Yaskawa INFORM job: X2_29-32(-90,180).JBI

/JOB
//NAME X2_29-32(-90,180)
//POS
///NPOS 300,300,300,19,0,0
///TOOL 0
///POSTYPE PULSE
///PULSE
C00000=2000,-95440,-72516,0,38121,0
C00001=-80443,-95440,-72516,-46202,38121,50067
C00002=-52411,-63190,-65629,-41206,65263,51508
C00003=-73087,-23788,-54178,-20049,70640,39353
C00004=-137855,-58890,-63164,50426,57117,3007
C00005=-121629,-1819,-23267,32035,72941,16834
C00006=-120935,3126,-16373,32060,71231,16611
C00007=-120668,5150,-13541,32087,70531,16512
C00008=-120826,7275,-11699,32150,70554,16454
C00009=-120668,5150,-13541,32087,70531,16512
C00010=-120649,6560,-12069,32112,70369,16472
C00011=-120645,6560,-10825,32251,69714,16277
C00012=-120649,6560,-12069,32112,70369,16472
C00013=-120913,4529,-14922,32082,71075,16573
C00014=-121602,-429,-21862,32048,72802,16805
C00015=-120074,-1541,-23154,10906,71264,22392
C00016=-120462,3262,-16191,11181,69532,22093
C00017=-120612,5232,-13331,11295,68818,21971
C00018=-120770,7357,-11488,11363,68799,21912
C00019=-120612,5232,-13331,11295,68818,21971
C00020=-120702,6360,-12382,11332,68826,21940
C00021=-120699,6356,-11141,11388,68075,21868
C00022=-120702,6360,-12382,11332,68826,21940
C00023=-120555,4389,-15254,11219,69547,22062
C00024=-120172,-412,-22245,10944,71297,22361
C00025=-119941,-49108,-60020,12756,52739,20459
C00026=-119789,-74783,-79746,11606,60570,21449
C00027=-121427,-115493,-86071,-971,23186,13
C00028=-103613,-33005,-61039,-35202,65094,-22685
C00029=-118652,-1130,-18887,-50959,75871,-22344
C00030=-120065,3095,-12579,-50928,73991,-22034
C00031=-120612,5858,-10323,-50783,73711,-22168
C00032=-120794,7716,-8707,-50742,73586,-22192
C00033=-120612,6719,-9575,-50786,73699,-22162
C00034=-120612,6754,-8612,-50907,73330,-21953
C00035=-120612,6719,-9575,-50786,73699,-22162
C00036=-120164,4326,-11494,-50910,73914,-22043
C00037=-118762,92,-17836,-50934,75798,-22362
C00038=-120082,-2017,-23568,-21020,76850,-12939
C00039=-120471,2786,-16617,-21041,75059,-12760
C00040=-120621,6055,-13261,-21027,74660,-12744
C00041=-120866,7545,-11965,-20950,74569,-12818
C00042=-120698,6523,-12855,-21003,74632,-12768
C00043=-120698,6506,-12245,-21039,74273,-12705
C00044=-120698,6523,-12855,-21003,74632,-12768
C00045=-120547,3972,-15593,-21018,75020,-12781
C00046=-120163,-831,-22574,-20994,76828,-12964
C00047=-120068,-2141,-23641,-4094,79360,4817
C00048=-120458,2664,-16692,-4000,77538,4745
C00049=-120609,5664,-13523,-3960,77123,4708
C00050=-120915,7025,-12341,-3868,77081,4605
C00051=-120609,5664,-13523,-3960,77123,4708
C00052=-120609,5646,-12752,-3962,76640,4725
C00053=-120609,5664,-13523,-3960,77123,4708
C00054=-120559,4206,-15421,-3970,77544,4711
C00055=-120175,-595,-22406,-4061,79389,4780
C00056=-120687,14813,-21149,-8531,87328,5298
C00057=-120686,13947,-18988,-8540,85572,5418
C00058=-121162,15330,-17687,-8405,85435,5272
C00059=-120827,14308,-18485,-8500,85444,5381
C00060=-120926,18777,-11948,-23218,84672,-11491
C00061=-120686,12805,-15419,-25390,80631,-12632
C00062=-120686,13423,-17789,-25296,82244,-12980
C00063=-103613,-33005,-61039,-35202,65094,-22685
C00064=-121427,-115493,-86071,-971,23186,13
C00065=-119789,-74783,-79746,11606,60570,21449
C00066=-119941,-49108,-60020,12756,52739,20459
C00067=-120686,14413,-19191,15888,76861,21657
C00068=-120686,13677,-16924,15998,75153,21431
C00069=-120864,13854,-15557,16118,74464,21280
C00070=-120686,13319,-15964,16052,74414,21331
C00071=-120685,12972,2532,58159,63782,21773
C00072=-120685,12849,1627,57961,64053,21984
C00073=-120685,12557,-1021,57383,64873,22611
C00074=-118042,2496,-28680,21493,77866,23942
C00075=-119941,-49108,-60020,12756,52739,20459
C00076=-119789,-74783,-79746,11606,60570,21449
C00077=-121427,-115493,-86071,-971,23186,13
C00078=-103613,-33005,-61039,-35202,65094,-22685
C00079=-134099,37898,13128,-30528,62935,-29291
C00080=-134100,37844,14655,-30775,62096,-29040
C00081=-131820,39720,18358,-33617,61933,-27865
C00082=-133865,38946,16955,-31235,61462,-28734
C00083=-133724,38989,23896,-55752,81870,-5528
C00084=-134106,38309,22847,-57056,83615,-3951
C00085=-130543,37429,19989,-57378,86491,-3781
C00086=-124532,-28339,-37080,2656,37858,63256
C00087=-80443,-95440,-72516,-46202,38121,50067
C00088=-628,-74499,-67639,-57475,89722,72456
C00089=3643,-76224,-106676,19950,71810,76872
C00090=-57022,-39792,-97587,-14580,73098,62715
C00091=-77894,6609,-39652,-10081,68656,55583
C00092=-79326,8848,-34628,-9340,66588,55287
C00093=-79882,9812,-32559,-9051,65763,55166
C00094=-80655,11957,-30643,-8578,65611,54918
C00095=-79882,9812,-32559,-9051,65763,55166
C00096=-80541,11612,-30977,-8647,65649,54954
C00097=-80539,10894,-29907,-8717,64633,55031
C00098=-80541,11612,-30977,-8647,65649,54954
C00099=-79996,10638,-33064,-8931,66478,55073
C00100=-78593,8374,-38132,-9661,68553,55366
C00101=-77879,6415,-39661,-10096,68566,55596
C00102=-79312,8664,-34633,-9354,66499,55298
C00103=-79868,9631,-32562,-9065,65674,55178
C00104=-80642,11778,-30647,-8592,65523,54929
C00105=-79868,9631,-32562,-9065,65674,55178
C00106=-80486,11377,-31039,-8686,65573,54978
C00107=-80483,10662,-29965,-8757,64557,55056
C00108=-80486,11377,-31039,-8686,65573,54978
C00109=-79940,10400,-33127,-8971,66401,55097
C00110=-78534,8129,-38197,-9702,68474,55392
C00111=-80101,2636,-42462,-8765,68121,54914
C00112=-81514,5018,-37368,-8012,66098,54596
C00113=-82062,6036,-35274,-7718,65291,54467
C00114=-82824,8247,-33345,-7247,65177,54218
C00115=-82062,6036,-35274,-7718,65291,54467
C00116=-82687,7884,-33751,-7328,65251,54260
C00117=-82684,7173,-32662,-7390,64223,54326
C00118=-82687,7884,-33751,-7328,65251,54260
C00119=-82150,6860,-35861,-7618,66062,54387
C00120=-80765,4464,-40992,-8359,68092,54701
C00121=-102565,-17528,-58279,5105,67037,47705
C00122=-103540,-14129,-52689,5779,65410,47308
C00123=-103914,-12731,-50412,6044,64755,47149
C00124=-104433,-9984,-48291,6364,64897,46981
C00125=-103914,-12731,-50412,6044,64755,47149
C00126=-104359,-10402,-48741,6314,64954,47009
C00127=-104354,-11138,-47602,6366,63880,46952
C00128=-104359,-10402,-48741,6314,64954,47009
C00129=-103995,-11787,-51026,6054,65619,47167
C00130=-103047,-15149,-56634,5395,67274,47560
C00131=-80233,11979,-33534,-13378,69985,55632
C00132=-80229,10556,-31784,-13533,68226,55836
C00133=-80227,10062,-31089,-13596,67561,55913
C00134=-85904,3072,-37201,-10254,66968,54061
C00135=-91604,-2565,-41777,-6847,66341,52198
C00136=-101176,-9655,-47350,-1032,65699,49019
C00137=-100886,-9155,-48096,-1203,66417,49108
C00138=-100216,-7271,-49632,-1590,68341,49304
C00139=-80300,11336,-32181,-3939,63811,54132
C00140=-80297,10024,-30348,-4003,62013,54196
C00141=-80296,9579,-29637,-4028,61349,54220
C00142=-80356,9883,-29495,-3999,61418,54197
C00143=-80338,10281,-30338,-3972,62137,54177
C00144=-80341,11605,-32161,-3909,63935,54114
C00145=-57022,-39792,-97587,-14580,73098,62715
C00146=-628,-74499,-67639,-57475,89722,72456
C00147=-628,-74499,-67639,-57475,89722,72456
C00148=-616,-75233,-71189,-57531,90735,71761
C00149=3643,-76224,-106674,19950,71813,76873
C00150=-42730,11015,-70691,-38334,96086,2936
C00151=-63606,9545,-60534,-45336,92087,-16638
C00152=-78956,5069,-41799,-36523,82652,-30708
C00153=-79715,8164,-36018,-36343,80767,-30358
C00154=-80007,9457,-33651,-36288,80012,-30216
C00155=-80417,12097,-31285,-36126,79775,-30292
C00156=-80007,9457,-33651,-36288,80012,-30216
C00157=-80344,11698,-31669,-36153,79828,-30282
C00158=-80337,10939,-30633,-36254,78993,-30001
C00159=-80344,11698,-31669,-36153,79828,-30282
C00160=-80059,10405,-34052,-36203,80590,-30428
C00161=-79319,7312,-39869,-36371,82488,-30786
C00162=-78994,5332,-41692,-36502,82694,-30736
C00163=-79751,8420,-35912,-36322,80808,-30385
C00164=-80043,9710,-33546,-36267,80051,-30242
C00165=-80452,12349,-31177,-36105,79813,-30317
C00166=-80043,9710,-33546,-36267,80051,-30242
C00167=-80378,11838,-31671,-36133,79874,-30310
C00168=-80371,11075,-30637,-36233,79039,-30029
C00169=-80378,11838,-31671,-36133,79874,-30310
C00170=-80093,10547,-34052,-36183,80637,-30456
C00171=-79355,7462,-39866,-36352,82536,-30815
C00172=-79090,5824,-41546,-36452,82791,-30803
C00173=-79842,8894,-35770,-36272,80900,-30451
C00174=-80133,10177,-33405,-36216,80142,-30307
C00175=-80539,12815,-31031,-36055,79902,-30380
C00176=-80133,10177,-33405,-36216,80142,-30307
C00177=-80467,12378,-31515,-36079,79989,-30382
C00178=-80461,11606,-30490,-36178,79153,-30101
C00179=-80467,12378,-31515,-36079,79989,-30382
C00180=-80184,11095,-33894,-36130,80753,-30529
C00181=-79450,8031,-39703,-36300,82657,-30890
C00182=-79130,5997,-41490,-36432,82820,-30827
C00183=-79881,9061,-35715,-36251,80928,-30474
C00184=-80171,10342,-33350,-36196,80169,-30330
C00185=-80577,12980,-30974,-36035,79928,-30403
C00186=-80171,10342,-33350,-36196,80169,-30330
C00187=-80499,12601,-31443,-36059,80034,-30409
C00188=-80493,11826,-30422,-36158,79199,-30129
C00189=-80499,12601,-31443,-36059,80034,-30409
C00190=-80216,11321,-33822,-36110,80799,-30556
C00191=-79484,8265,-39628,-36281,82705,-30918
C00192=-80360,13355,-34008,-31162,79863,-31191
C00193=-80358,11846,-32319,-31320,78301,-30757
C00194=-80129,11573,-31352,-31494,77744,-30518
C00195=-80458,11751,-31298,-31342,77685,-30622
C00196=-80398,12063,-32232,-31297,78337,-30782
C00197=-80400,13577,-33916,-31139,79899,-31215
C00198=-80289,11819,-32883,-40833,82428,-30239
C00199=-80286,10439,-31086,-40975,81039,-29694
C00200=-80284,9940,-30341,-41041,80492,-29477
C00201=-80262,9799,-30343,-41055,80447,-29451
C00202=-80245,10226,-31168,-40996,81011,-29666
C00203=-80248,11601,-32971,-40853,82401,-30212
C00204=-66712,19655,-58640,-43457,90055,-24381
C00205=-33423,17994,-60377,-60627,102988,-19600
C00206=-628,-74499,-67639,-57475,89722,-77289
C00207=-111516,-94989,-87682,-11539,41033,-8318
C00208=-107125,-12532,-46236,-32676,64375,-10703
C00209=-119952,37605,6162,-31233,75137,-17424
C00210=-120511,42562,14108,-31354,72919,-17016
C00211=-120728,44654,17433,-31427,72005,-16841
C00212=-120598,46946,19889,-31526,71766,-16719
C00213=-120728,44654,17433,-31427,72005,-16841
C00214=-120690,45788,18679,-31469,71861,-16784
C00215=-120687,45721,19851,-31594,71213,-16595
C00216=-120690,45788,18679,-31469,71861,-16784
C00217=-120474,43679,15324,-31394,72783,-16962
C00218=-119917,38688,7316,-31265,75018,-17376
C00219=-121235,29127,929,-10497,72605,-22385
C00220=-120892,33963,8709,-10768,70384,-22067
C00221=-120760,35995,11952,-10883,69467,-21936
C00222=-120625,38237,14258,-10956,69222,-21864
C00223=-120760,35995,11952,-10883,69467,-21936
C00224=-120657,37146,13206,-10937,69303,-21884
C00225=-120654,37124,14427,-10991,68554,-21813
C00226=-120657,37146,13206,-10937,69303,-21884
C00227=-120788,35099,9935,-10821,70230,-22016
C00228=-121127,30229,2096,-10548,72470,-22335
C00229=-114017,-48711,-62992,-16459,47417,-13874
C00230=-111516,-94989,-87682,-11539,41033,-8318
C00231=-126605,-77887,-93073,32833,63422,15189
C00232=-122507,12852,-43627,17515,100315,22769
C00233=-122731,-562,-19309,51196,76332,22742
C00234=-121309,3590,-13049,51151,74446,22427
C00235=-120759,5312,-10468,51156,73690,22291
C00236=-120602,7442,-8613,51127,73573,22309
C00237=-120759,5312,-10468,51156,73690,22291
C00238=-120666,6547,-9361,51143,73609,22295
C00239=-120662,6597,-8073,51308,73115,22013
C00240=-120666,6547,-9361,51143,73609,22295
C00241=-121212,4820,-11958,51134,74367,22434
C00242=-122622,659,-18251,51172,76257,22758
C00243=-122507,10859,-42333,17402,98575,22516
C00244=-121302,-1391,-23074,21379,77148,13095
C00245=-120901,3377,-16122,21398,75339,12912
C00246=-120747,5333,-13267,21416,74597,12833
C00247=-120590,7459,-11416,21370,74514,12875
C00248=-120747,5333,-13267,21416,74597,12833
C00249=-120673,6521,-12221,21396,74547,12851
C00250=-120670,6504,-10992,21468,73832,12721
C00251=-120673,6521,-12221,21396,74547,12851
C00252=-120826,4563,-15090,21376,75296,12931
C00253=-121222,-206,-22073,21354,77121,13119
C00254=-121314,-1652,-23262,4485,79740,-4708
C00255=-120913,3117,-16316,4391,77900,-4639
C00256=-120758,5074,-13462,4356,77144,-4613
C00257=-120601,7199,-11615,4311,77090,-4561
C00258=-120758,5074,-13462,4356,77144,-4613
C00259=-120661,6618,-12165,4328,77134,-4580
C00260=-120658,6600,-10936,4339,76370,-4606
C00261=-120661,6618,-12165,4328,77134,-4580
C00262=-120814,4660,-15035,4362,77900,-4605
C00263=-121209,-107,-22019,4454,79763,-4672
C00264=-120687,46979,12625,8958,83453,-5452
C00265=-120687,46939,12852,8960,83294,-5464
C00266=-121610,47377,14332,9229,82719,-5809
C00267=-120687,46779,13614,8967,82756,-5503
C00268=-120687,46744,18453,25999,77793,12121
C00269=-120687,46348,16793,25935,78533,12285
C00270=-120687,46750,14296,25811,80109,12635
C00271=-133650,-5326,-40947,35821,67459,4738
C00272=-126605,-79487,-84548,34660,58331,13454
C00273=-111516,-94989,-87682,-11539,41033,-8318
C00274=-114017,-48711,-62992,-16459,47417,-13874
C00275=-117875,8541,-26754,-15356,68464,-18868
C00276=-120687,46680,12303,-15684,74586,-21239
C00277=-120687,46183,14573,-15804,72993,-21028
C00278=-120687,45847,15503,-15862,72274,-20933
C00279=-120687,45820,15711,-15860,72146,-20914
C00280=-120686,46430,31549,-51889,62431,-21622
C00281=-120686,46225,30262,-51616,62867,-21897
C00282=-120686,45862,27317,-50999,63909,-22538
C00283=-117875,8541,-26754,-15356,68464,-18868
C00284=-114017,-48711,-62992,-16459,47417,-13874
C00285=-111516,-94989,-87682,-11539,41033,-8318
C00286=-126605,-79487,-84548,34660,58331,13454
C00287=-133650,-5326,-40947,35821,67459,4738
C00288=-107292,16964,-8341,30286,65218,30077
C00289=-107291,16711,-5651,30703,63668,29626
C00290=-107319,17056,-4163,30899,63039,29427
C00291=-107325,17150,-4064,30903,63037,29424
C00292=-107531,17120,3962,56911,83437,5110
C00293=-107292,16975,3345,57479,84239,4502
C00294=-107292,16775,1094,57407,84952,4997
C00295=-118083,23631,-28824,25815,115568,5891
C00296=-116334,-45445,-82386,24519,90130,1359
C00297=-114916,-111439,-107393,23774,54945,-5331
C00298=-628,-74499,-67639,-57475,89722,-77289
C00299=2000,17994,-60377,0,102988,0
BC00000=30861,666204,744559
BC00001=125925,693938,117612
BC00002=171995,715848,96803
BC00003=199966,729151,84169
BC00004=289373,771673,43785
BC00005=289373,771673,43785
BC00006=289373,771673,43785
BC00007=289373,771673,43785
BC00008=289373,771673,43785
BC00009=289373,771673,43785
BC00010=289373,771673,43785
BC00011=289373,771673,43785
BC00012=289373,771673,43785
BC00013=289373,771673,43785
BC00014=289373,771673,43785
BC00015=275430,758658,78312
BC00016=275430,758658,78312
BC00017=275430,758658,78312
BC00018=275430,758658,78312
BC00019=275430,758658,78312
BC00020=275430,758658,78312
BC00021=275430,758658,78312
BC00022=275430,758658,78312
BC00023=275430,758658,78312
BC00024=275430,758658,78312
BC00025=275430,725446,78312
BC00026=275430,674753,78312
BC00027=160005,679271,117612
BC00028=134493,734471,53
BC00029=134493,734471,53
BC00030=134493,734471,53
BC00031=134493,734471,53
BC00032=134493,734471,53
BC00033=134493,734471,53
BC00034=134493,734471,53
BC00035=134493,734471,53
BC00036=134493,734471,53
BC00037=134493,734471,53
BC00038=120013,731989,63282
BC00039=120013,731989,63282
BC00040=120013,731989,63282
BC00041=120013,731989,63282
BC00042=120013,731989,63282
BC00043=120013,731989,63282
BC00044=120013,731989,63282
BC00045=120013,731989,63282
BC00046=120013,731989,63282
BC00047=143296,743099,87341
BC00048=143296,743099,87341
BC00049=143296,743099,87341
BC00050=143296,743099,87341
BC00051=143296,743099,87341
BC00052=143296,743099,87341
BC00053=143296,743099,87341
BC00054=143296,743099,87341
BC00055=143296,743099,87341
BC00056=160875,733218,0
BC00057=159215,738452,0
BC00058=159050,738970,0
BC00059=154263,739676,0
BC00060=124438,729775,0
BC00061=121804,726587,0
BC00062=123464,721353,0
BC00063=134493,734471,53
BC00064=160005,679271,117612
BC00065=275430,674753,78312
BC00066=275430,725446,78312
BC00067=261630,745054,0
BC00068=261335,750526,0
BC00069=262635,752963,0
BC00070=310200,761264,0
BC00071=269037,768534,0
BC00072=267560,766459,0
BC00073=263869,761272,0
BC00074=263869,761272,0
BC00075=275430,725446,78312
BC00076=275430,674753,78312
BC00077=160005,679271,117612
BC00078=134493,734471,53
BC00079=177141,688062,0
BC00080=175480,693296,0
BC00081=174817,695179,178
BC00082=160472,692881,15
BC00083=152915,732429,1
BC00084=154775,734615,0
BC00085=161011,731782,0
BC00086=160005,693938,117612
BC00087=125925,693938,117612
BC00088=97174,666880,426359
BC00089=199464,674570,1075173
BC00090=48447,721710,1061717
BC00091=196183,770700,1075175
BC00092=196183,770700,1075175
BC00093=196183,770700,1075175
BC00094=196183,770700,1075175
BC00095=196183,770700,1075175
BC00096=196183,770700,1075175
BC00097=196183,770700,1075175
BC00098=196183,770700,1075175
BC00099=196183,770700,1075175
BC00100=196183,770700,1075175
BC00101=139869,760824,1075175
BC00102=139869,760824,1075175
BC00103=139869,760824,1075175
BC00104=139869,760824,1075175
BC00105=139869,760824,1075175
BC00106=139869,760824,1075175
BC00107=139869,760824,1075175
BC00108=139869,760824,1075175
BC00109=139869,760824,1075175
BC00110=139869,760824,1075175
BC00111=15,735270,1075175
BC00112=15,735270,1075175
BC00113=15,735270,1075175
BC00114=15,735270,1075175
BC00115=15,735270,1075175
BC00116=15,735270,1075175
BC00117=15,735270,1075175
BC00118=15,735270,1075175
BC00119=15,735270,1075175
BC00120=15,735270,1075175
BC00121=15,725270,1075175
BC00122=15,725270,1075175
BC00123=15,725270,1075175
BC00124=15,725270,1075175
BC00125=15,725270,1075175
BC00126=15,725270,1075175
BC00127=15,725270,1075175
BC00128=15,725270,1075175
BC00129=15,725270,1075175
BC00130=15,725270,1075175
BC00131=12536,730414,1075175
BC00132=10876,735648,1075175
BC00133=10211,737741,1075175
BC00134=7204,734292,1075175
BC00135=4400,731075,1075175
BC00136=15,726043,1075175
BC00137=15,723950,1075175
BC00138=15,718716,1075175
BC00139=125627,754347,1075175
BC00140=125333,759820,1075175
BC00141=125215,762009,1075175
BC00142=192338,773707,1075173
BC00143=192456,771518,1075175
BC00144=192751,766045,1075175
BC00145=48447,721710,1061717
BC00146=97174,666880,1005640
BC00147=97174,666880,842388
BC00148=97174,666880,900747
BC00149=199464,674570,1075172
BC00150=79996,736581,994878
BC00151=45352,753605,1043201
BC00152=33984,772629,1075175
BC00153=33984,772629,1075175
BC00154=33984,772629,1075175
BC00155=33984,772629,1075175
BC00156=33984,772629,1075175
BC00157=33984,772629,1075175
BC00158=33984,772629,1075175
BC00159=33984,772629,1075175
BC00160=33984,772629,1075175
BC00161=33984,772629,1075175
BC00162=90316,762849,1075175
BC00163=90316,762849,1075175
BC00164=90316,762849,1075175
BC00165=90316,762849,1075175
BC00166=90316,762849,1075175
BC00167=90316,762849,1075175
BC00168=90316,762849,1075175
BC00169=90316,762849,1075175
BC00170=90316,762849,1075175
BC00171=90316,762849,1075175
BC00172=237131,737545,1075175
BC00173=237131,737545,1075175
BC00174=237131,737545,1075175
BC00175=237131,737545,1075175
BC00176=237131,737545,1075175
BC00177=237131,737545,1075175
BC00178=237131,737545,1075175
BC00179=237131,737545,1075175
BC00180=237131,737545,1075175
BC00181=237131,737545,1075175
BC00182=294635,727643,1075175
BC00183=294635,727643,1075175
BC00184=294635,727643,1075175
BC00185=294635,727643,1075175
BC00186=294635,727643,1075175
BC00187=294635,727643,1075175
BC00188=294635,727643,1075175
BC00189=294635,727643,1075175
BC00190=294635,727643,1075175
BC00191=294635,727643,1075175
BC00192=217651,732700,1075175
BC00193=219347,737901,1075175
BC00194=220025,739981,1075175
BC00195=287170,728397,1075175
BC00196=286492,726316,1075175
BC00197=284797,721115,1075175
BC00198=104549,756414,1075175
BC00199=104877,761851,1075175
BC00200=105009,764026,1075175
BC00201=37863,775610,1075175
BC00202=37732,773435,1075175
BC00203=37403,767998,1075175
BC00204=32590,750193,986570
BC00205=32590,674533,986570
BC00206=97174,666880,426359
BC00207=147937,670008,53
BC00208=147937,711773,53
BC00209=147937,730150,53
BC00210=147937,730150,53
BC00211=147937,730150,53
BC00212=147937,730150,53
BC00213=147937,730150,53
BC00214=147937,730150,53
BC00215=147937,730150,53
BC00216=147937,730150,53
BC00217=147937,730150,53
BC00218=147937,730150,53
BC00219=158165,726651,59010
BC00220=158165,726651,59010
BC00221=158165,726651,59010
BC00222=158165,726651,59010
BC00223=158165,726651,59010
BC00224=158165,726651,59010
BC00225=158165,726651,59010
BC00226=158165,726651,59010
BC00227=158165,726651,59010
BC00228=158165,726651,59010
BC00229=154158,704461,35913
BC00230=147937,670008,53
BC00231=303968,673866,53
BC00232=303968,733345,53
BC00233=303968,733345,53
BC00234=303968,733345,53
BC00235=303968,733345,53
BC00236=303968,733345,53
BC00237=303968,733345,53
BC00238=303968,733345,53
BC00239=303968,733345,53
BC00240=303968,733345,53
BC00241=303968,733345,53
BC00242=303968,733345,53
BC00243=303968,733345,53
BC00244=317859,731237,70095
BC00245=317859,731237,70095
BC00246=317859,731237,70095
BC00247=317859,731237,70095
BC00248=317859,731237,70095
BC00249=317859,731237,70095
BC00250=317859,731237,70095
BC00251=317859,731237,70095
BC00252=317859,731237,70095
BC00253=317859,731237,70095
BC00254=294346,742753,94560
BC00255=294346,742753,94560
BC00256=294346,742753,94560
BC00257=294346,742753,94560
BC00258=294346,742753,94560
BC00259=294346,742753,94560
BC00260=294346,742753,94560
BC00261=294346,742753,94560
BC00262=294346,742753,94560
BC00263=294346,742753,94560
BC00264=276740,698523,17248
BC00265=278435,703724,53
BC00266=279113,705804,53
BC00267=283819,705005,53
BC00268=316764,693534,53
BC00269=316086,691453,53
BC00270=314391,686252,53
BC00271=314391,686252,53
BC00272=303968,673866,53
BC00273=147937,670008,53
BC00274=154158,704461,35913
BC00275=166916,707890,15720
BC00276=176272,710404,912
BC00277=176601,715841,53
BC00278=176732,718016,53
BC00279=127735,726480,51
BC00280=162022,730813,53
BC00281=163238,728692,53
BC00282=166278,723391,53
BC00283=166916,707890,15720
BC00284=154158,704461,35913
BC00285=147937,670008,53
BC00286=303968,673866,53
BC00287=314391,686252,53
BC00288=265210,708896,0
BC00289=266905,714097,0
BC00290=267584,716178,0
BC00291=283264,713482,0
BC00292=289747,755484,0
BC00293=287471,755837,0
BC00294=281210,753020,0
BC00295=281210,753020,0
BC00296=281210,753020,0
BC00297=281210,753020,0
BC00298=97174,666880,426359
BC00299=32590,674533,986570
EC00000=-798156,1112951
EC00001=-798156,1112951
EC00002=-798156,1112951
EC00003=-798156,1112951
EC00004=-798156,1112951
EC00005=-798156,1112951
EC00006=-798156,1112951
EC00007=-798156,1112951
EC00008=-798156,1112951
EC00009=-798156,1112951
EC00010=-798156,1112951
EC00011=-798156,1112951
EC00012=-798156,1112951
EC00013=-798156,1112951
EC00014=-798156,1112951
EC00015=-798156,1112951
EC00016=-798156,1112951
EC00017=-798156,1112951
EC00018=-798156,1112951
EC00019=-798156,1112951
EC00020=-798156,1112951
EC00021=-798156,1112951
EC00022=-798156,1112951
EC00023=-798156,1112951
EC00024=-798156,1112951
EC00025=-798156,1112951
EC00026=-798156,1112951
EC00027=-798156,1112951
EC00028=-798156,1112951
EC00029=-798156,1112951
EC00030=-798156,1112951
EC00031=-798156,1112951
EC00032=-798156,1112951
EC00033=-798156,1112951
EC00034=-798156,1112951
EC00035=-798156,1112951
EC00036=-798156,1112951
EC00037=-798156,1112951
EC00038=-798156,1112951
EC00039=-798156,1112951
EC00040=-798156,1112951
EC00041=-798156,1112951
EC00042=-798156,1112951
EC00043=-798156,1112951
EC00044=-798156,1112951
EC00045=-798156,1112951
EC00046=-798156,1112951
EC00047=-798156,1112951
EC00048=-798156,1112951
EC00049=-798156,1112951
EC00050=-798156,1112951
EC00051=-798156,1112951
EC00052=-798156,1112951
EC00053=-798156,1112951
EC00054=-798156,1112951
EC00055=-798156,1112951
EC00056=-798156,1112951
EC00057=-798156,1112951
EC00058=-798156,1112951
EC00059=-798156,1112951
EC00060=-798156,1112951
EC00061=-798156,1112951
EC00062=-798156,1112951
EC00063=-798156,1112951
EC00064=-798156,1112951
EC00065=-798156,1112951
EC00066=-798156,1112951
EC00067=-798156,1112951
EC00068=-798156,1112951
EC00069=-798156,1112951
EC00070=-798156,1112951
EC00071=-798156,1112951
EC00072=-798156,1112951
EC00073=-798156,1112951
EC00074=-798156,1112951
EC00075=-798156,1112951
EC00076=-798156,1112951
EC00077=-798156,1112951
EC00078=-798156,1112951
EC00079=-798156,1112951
EC00080=-798156,1112951
EC00081=-798155,1112951
EC00082=-798156,1112951
EC00083=-798156,1112951
EC00084=-798156,1112951
EC00085=-798156,1112951
EC00086=-798156,1112951
EC00087=-798156,1112951
EC00088=-798156,1112951
EC00089=-798156,1112951
EC00090=-798156,1112951
EC00091=-798156,1112951
EC00092=-798156,1112951
EC00093=-798156,1112951
EC00094=-798156,1112951
EC00095=-798156,1112951
EC00096=-798156,1112951
EC00097=-798156,1112951
EC00098=-798156,1112951
EC00099=-798156,1112951
EC00100=-798156,1112951
EC00101=-798156,1112951
EC00102=-798156,1112951
EC00103=-798156,1112951
EC00104=-798156,1112951
EC00105=-798156,1112951
EC00106=-798156,1112951
EC00107=-798156,1112951
EC00108=-798156,1112951
EC00109=-798156,1112951
EC00110=-798156,1112951
EC00111=-798156,1112951
EC00112=-798156,1112951
EC00113=-798156,1112951
EC00114=-798156,1112951
EC00115=-798156,1112951
EC00116=-798156,1112951
EC00117=-798156,1112951
EC00118=-798156,1112951
EC00119=-798156,1112951
EC00120=-798156,1112951
EC00121=-798156,1112951
EC00122=-798156,1112951
EC00123=-798156,1112951
EC00124=-798156,1112951
EC00125=-798156,1112951
EC00126=-798156,1112951
EC00127=-798156,1112951
EC00128=-798156,1112951
EC00129=-798156,1112951
EC00130=-798156,1112951
EC00131=-798156,1112951
EC00132=-798156,1112951
EC00133=-798156,1112951
EC00134=-798156,1112951
EC00135=-798156,1112951
EC00136=-798156,1112951
EC00137=-798156,1112951
EC00138=-798156,1112951
EC00139=-798156,1112951
EC00140=-798156,1112951
EC00141=-798156,1112951
EC00142=-798155,1112951
EC00143=-798156,1112951
EC00144=-798156,1112951
EC00145=-798156,1112951
EC00146=-798156,1112951
EC00147=-850885,799301
EC00148=-850885,361850
EC00149=-798154,-3
EC00150=-798156,0
EC00151=-798156,0
EC00152=-798156,0
EC00153=-798156,0
EC00154=-798156,0
EC00155=-798156,0
EC00156=-798156,0
EC00157=-798156,0
EC00158=-798156,0
EC00159=-798156,0
EC00160=-798156,0
EC00161=-798156,0
EC00162=-798156,0
EC00163=-798156,0
EC00164=-798156,0
EC00165=-798156,0
EC00166=-798156,0
EC00167=-798156,0
EC00168=-798156,0
EC00169=-798156,0
EC00170=-798156,0
EC00171=-798156,0
EC00172=-798156,0
EC00173=-798156,0
EC00174=-798156,0
EC00175=-798156,0
EC00176=-798156,0
EC00177=-798156,0
EC00178=-798156,0
EC00179=-798156,0
EC00180=-798156,0
EC00181=-798156,0
EC00182=-798156,0
EC00183=-798156,0
EC00184=-798156,0
EC00185=-798156,0
EC00186=-798156,0
EC00187=-798156,0
EC00188=-798156,0
EC00189=-798156,0
EC00190=-798156,0
EC00191=-798156,0
EC00192=-798156,0
EC00193=-798156,0
EC00194=-798156,0
EC00195=-798156,0
EC00196=-798156,0
EC00197=-798156,0
EC00198=-798156,0
EC00199=-798156,0
EC00200=-798156,0
EC00201=-798156,0
EC00202=-798156,0
EC00203=-798156,0
EC00204=-798156,0
EC00205=-798156,0
EC00206=-798156,0
EC00207=-798156,0
EC00208=-798156,0
EC00209=-798156,0
EC00210=-798156,0
EC00211=-798156,0
EC00212=-798156,0
EC00213=-798156,0
EC00214=-798156,0
EC00215=-798156,0
EC00216=-798156,0
EC00217=-798156,0
EC00218=-798156,0
EC00219=-798156,0
EC00220=-798156,0
EC00221=-798156,0
EC00222=-798156,0
EC00223=-798156,0
EC00224=-798156,0
EC00225=-798156,0
EC00226=-798156,0
EC00227=-798156,0
EC00228=-798156,0
EC00229=-798156,0
EC00230=-798156,0
EC00231=-798156,0
EC00232=-798156,0
EC00233=-798156,0
EC00234=-798156,0
EC00235=-798156,0
EC00236=-798156,0
EC00237=-798156,0
EC00238=-798156,0
EC00239=-798156,0
EC00240=-798156,0
EC00241=-798156,0
EC00242=-798156,0
EC00243=-798156,0
EC00244=-798156,0
EC00245=-798156,0
EC00246=-798156,0
EC00247=-798156,0
EC00248=-798156,0
EC00249=-798156,0
EC00250=-798156,0
EC00251=-798156,0
EC00252=-798156,0
EC00253=-798156,0
EC00254=-798156,0
EC00255=-798156,0
EC00256=-798156,0
EC00257=-798156,0
EC00258=-798156,0
EC00259=-798156,0
EC00260=-798156,0
EC00261=-798156,0
EC00262=-798156,0
EC00263=-798156,0
EC00264=-798156,0
EC00265=-798156,0
EC00266=-798156,0
EC00267=-798156,0
EC00268=-798156,0
EC00269=-798156,0
EC00270=-798156,0
EC00271=-798156,0
EC00272=-798156,0
EC00273=-798156,0
EC00274=-798156,0
EC00275=-798156,0
EC00276=-798156,0
EC00277=-798156,0
EC00278=-798156,0
EC00279=-798155,-1
EC00280=-798156,0
EC00281=-798156,0
EC00282=-798156,0
EC00283=-798156,0
EC00284=-798156,0
EC00285=-798156,0
EC00286=-798156,0
EC00287=-798156,0
EC00288=-798156,0
EC00289=-798156,0
EC00290=-798156,0
EC00291=-798156,0
EC00292=-798156,0
EC00293=-798156,0
EC00294=-798156,0
EC00295=-798156,0
EC00296=-798156,0
EC00297=-798156,0
EC00298=-798156,0
EC00299=-798156,0
///POSTYPE BASE
///RECTAN
///RCONF 0,0,0,0,0,0,0,0,0,0,0,0,0,0,0,0,0,0,0,0,0,0,0,0
P00006=0.222,-3.123,-1.508,0.0000,0.0000,0.0000
P00021=-0.225,-6.128,-0.405,0.0000,0.0000,0.0000
P00022=0.222,-3.123,-1.508,0.0000,0.0000,0.0000
P00023=0.143,-0.036,0.682,0.0000,0.0000,0.0000
P00024=0.145,-0.552,1.326,0.0000,0.0000,0.0000
P00025=-2.003,0.006,0.728,0.0000,0.0000,0.0000
P00026=0.562,-0.002,-0.337,0.0000,0.0000,0.0000
P00027=-0.746,0.015,-9.096,0.0000,0.0000,0.0000
P00028=-2.237,-0.018,-7.702,0.0000,0.0000,0.0000
///RCONF 0,0,0,0,1,0,0,0,0,0,0,0,0,0,0,0,0,0,0,0,0,0,0,0
P00033=-0.123,0.612,-5.012,0.0000,0.0000,0.0000
///RCONF 0,0,0,0,0,0,0,0,0,0,0,0,0,0,0,0,0,0,0,0,0,0,0,0
P00034=-0.304,0.773,-2.693,0.0000,0.0000,0.0000
P00035=2.817,0.591,-1.622,0.0000,0.0000,0.0000
P00036=-1.108,-0.829,1.850,0.0000,0.0000,0.0000
P00041=0.192,3.924,0.305,0.0000,0.0000,0.0000
P00042=-0.217,1.941,0.413,0.0000,0.0000,0.0000
P00043=-0.044,-1.937,1.197,0.0000,0.0000,0.0000
P00044=0.687,-2.322,1.156,0.0000,0.0000,0.0000
P00045=-0.068,-0.810,1.603,0.0000,0.0000,0.0000
P00046=0.799,0.043,1.292,0.0000,0.0000,0.0000
//INST
///DATE 2024/04/08 10:40
///ATTR SC,RW
///GROUP1 RB1,BS1
///GROUP2 ST1
NOP
'X2_29-32(-90,180)
MOVJ C00000 BC00000 VJ=100.00  +MOVJ EC00000 VJ=100.00
MOVJ C00001 BC00001 VJ=100.00  +MOVJ EC00001 VJ=100.00
MOVJ C00002 BC00002 VJ=100.00  +MOVJ EC00002 VJ=100.00
MOVJ C00003 BC00003 VJ=100.00  +MOVJ EC00003 VJ=100.00
MOVJ C00004 BC00004 VJ=100.00  +MOVJ EC00004 VJ=100.00
'Path S4862
SFTOF3D
MOVJ C00005 BC00005 VJ=100.00  +MOVJ EC00005 VJ=100.00
MOVL C00006 BC00006 V=800.0  +MOVJ EC00006 VJ=100.00
SMOVL C00007 BC00007 V=166.7  +MOVJ EC00007
SREFP 3 C00008 BC00008  +REFP EC00008
CALL JOB:SEARCH-R1-S13D
SET P042 P006
SFTON3D P042
SMOVL C00009 BC00009 V=166.7  +MOVJ EC00009
SMOVL C00010 BC00010 V=166.7  +MOVJ EC00010
SREFP 3 C00011 BC00011  +REFP EC00011
CALL JOB:SEARCH-R1-S13D
SET P042 P006
SFTON3D P042
SMOVL C00012 BC00012 V=166.7  +MOVJ EC00012
MOVL C00013 BC00013 V=800.0  +MOVJ EC00013 VJ=100.00
MOVL C00014 BC00014 V=1000.0  +MOVJ EC00014 VJ=100.00
'EndPath S4862
'Path S4863
SFTOF3D
MOVJ C00015 BC00015 VJ=100.00  +MOVJ EC00015 VJ=100.00
MOVL C00016 BC00016 V=800.0  +MOVJ EC00016 VJ=100.00
SMOVL C00017 BC00017 V=166.7  +MOVJ EC00017
SREFP 3 C00018 BC00018  +REFP EC00018
CALL JOB:SEARCH-R1-S13D
SET P041 P006
SFTON3D P041
SMOVL C00019 BC00019 V=166.7  +MOVJ EC00019
SMOVL C00020 BC00020 V=166.7  +MOVJ EC00020
SREFP 3 C00021 BC00021  +REFP EC00021
CALL JOB:SEARCH-R1-S13D
SET P041 P006
SFTON3D P041
SMOVL C00022 BC00022 V=166.7  +MOVJ EC00022
MOVL C00023 BC00023 V=800.0  +MOVJ EC00023 VJ=100.00
MOVL C00024 BC00024 V=1000.0  +MOVJ EC00024 VJ=100.00
'EndPath S4863
MOVJ C00025 BC00025 VJ=100.00  +MOVJ EC00025 VJ=100.00
MOVJ C00026 BC00026 VJ=100.00  +MOVJ EC00026 VJ=100.00
MOVJ C00027 BC00027 VJ=100.00  +MOVJ EC00027 VJ=100.00
MOVJ C00028 BC00028 VJ=100.00  +MOVJ EC00028 VJ=100.00
'Path S4864
SFTOF3D
MOVJ C00029 BC00029 VJ=100.00  +MOVJ EC00029 VJ=100.00
MOVL C00030 BC00030 V=800.0  +MOVJ EC00030 VJ=100.00
SMOVL C00031 BC00031 V=166.7  +MOVJ EC00031
SREFP 3 C00032 BC00032  +REFP EC00032
CALL JOB:SEARCH-R1-S13D
SET P045 P006
SFTON3D P045
SMOVL C00033 BC00033 V=166.7  +MOVJ EC00033
SREFP 3 C00034 BC00034  +REFP EC00034
CALL JOB:SEARCH-R1-S13D
SET P045 P006
SFTON3D P045
SMOVL C00035 BC00035 V=166.7  +MOVJ EC00035
MOVL C00036 BC00036 V=800.0  +MOVJ EC00036 VJ=100.00
MOVL C00037 BC00037 V=1000.0  +MOVJ EC00037 VJ=100.00
'EndPath S4864
'Path S4231
SFTOF3D
MOVJ C00038 BC00038 VJ=100.00  +MOVJ EC00038 VJ=100.00
MOVL C00039 BC00039 V=800.0  +MOVJ EC00039 VJ=100.00
SMOVL C00040 BC00040 V=166.7  +MOVJ EC00040
SREFP 3 C00041 BC00041  +REFP EC00041
CALL JOB:SEARCH-R1-S13D
SET P022 P006
SFTON3D P022
SMOVL C00042 BC00042 V=166.7  +MOVJ EC00042
SREFP 3 C00043 BC00043  +REFP EC00043
CALL JOB:SEARCH-R1-S13D
SET P022 P006
SFTON3D P022
SMOVL C00044 BC00044 V=166.7  +MOVJ EC00044
MOVL C00045 BC00045 V=800.0  +MOVJ EC00045 VJ=100.00
MOVL C00046 BC00046 V=1000.0  +MOVJ EC00046 VJ=100.00
'EndPath S4231
'Path S4232
SFTOF3D
MOVJ C00047 BC00047 VJ=100.00  +MOVJ EC00047 VJ=100.00
MOVL C00048 BC00048 V=800.0  +MOVJ EC00048 VJ=100.00
SMOVL C00049 BC00049 V=166.7  +MOVJ EC00049
SREFP 3 C00050 BC00050  +REFP EC00050
CALL JOB:SEARCH-R1-S13D
SET P021 P006
SFTON3D P021
SMOVL C00051 BC00051 V=166.7  +MOVJ EC00051
SREFP 3 C00052 BC00052  +REFP EC00052
CALL JOB:SEARCH-R1-S13D
SET P021 P006
SFTON3D P021
SMOVL C00053 BC00053 V=166.7  +MOVJ EC00053
MOVL C00054 BC00054 V=800.0  +MOVJ EC00054 VJ=100.00
MOVL C00055 BC00055 V=1000.0  +MOVJ EC00055 VJ=100.00
'EndPath S4232
'Path W4886
SFTOF3D
SFTON3D P021
MOVJ C00056 BC00056 VJ=100.00  +MOVJ EC00056 VJ=100.00
SMOVL C00057 BC00057 V=800.0  +MOVJ EC00057
SMOVL C00058 BC00058 V=150.0 PL=0  +MOVJ EC00058
MACRO1 MJ#(0) ARGF6
ARCON
SMOVL C00059 BC00059 V=8.3  +MOVJ EC00059
SFTON3D P022
SMOVL C00060 BC00060 V=8.3  +MOVJ EC00060
ARCOF
SMOVL C00061 BC00061 V=800.0  +MOVJ EC00061
SMOVL C00062 BC00062 V=1000.0  +MOVJ EC00062
SFTOF3D
'EndPath W4886
MOVJ C00063 BC00063 VJ=100.00  +MOVJ EC00063 VJ=100.00
MOVJ C00064 BC00064 VJ=100.00  +MOVJ EC00064 VJ=100.00
MOVJ C00065 BC00065 VJ=100.00  +MOVJ EC00065 VJ=100.00
MOVJ C00066 BC00066 VJ=100.00  +MOVJ EC00066 VJ=100.00
'Path W4887
SFTOF3D
SFTON3D P041
MOVJ C00067 BC00067 VJ=100.00  +MOVJ EC00067 VJ=100.00
SMOVL C00068 BC00068 V=800.0  +MOVJ EC00068
SMOVL C00069 BC00069 V=150.0 PL=0  +MOVJ EC00069
ARCON
SMOVL C00070 BC00070 V=8.3  +MOVJ EC00070
SFTON3D P042
SMOVL C00071 BC00071 V=8.3  +MOVJ EC00071
ARCOF
SMOVL C00072 BC00072 V=800.0  +MOVJ EC00072
SMOVL C00073 BC00073 V=1000.0  +MOVJ EC00073
SFTOF3D
'EndPath W4887
MOVJ C00074 BC00074 VJ=100.00  +MOVJ EC00074 VJ=100.00
MOVJ C00075 BC00075 VJ=100.00  +MOVJ EC00075 VJ=100.00
MOVJ C00076 BC00076 VJ=100.00  +MOVJ EC00076 VJ=100.00
MOVJ C00077 BC00077 VJ=100.00  +MOVJ EC00077 VJ=100.00
MOVJ C00078 BC00078 VJ=100.00  +MOVJ EC00078 VJ=100.00
'Path W4887
SFTOF3D
SFTON3D P045
MOVJ C00079 BC00079 VJ=100.00  +MOVJ EC00079 VJ=100.00
SMOVL C00080 BC00080 V=800.0  +MOVJ EC00080
SMOVL C00081 BC00081 V=150.0 PL=0  +MOVJ EC00081
ARCON
SMOVL C00082 BC00082 V=8.3  +MOVJ EC00082
SMOVL C00083 BC00083 V=8.3  +MOVJ EC00083
ARCOF
SMOVL C00084 BC00084 V=800.0  +MOVJ EC00084
SMOVL C00085 BC00085 V=1000.0  +MOVJ EC00085
SFTOF3D
'EndPath W4887
MOVJ C00086 BC00086 VJ=100.00  +MOVJ EC00086 VJ=100.00
MOVJ C00087 BC00087 VJ=100.00  +MOVJ EC00087 VJ=100.00
MOVJ C00088 BC00088 VJ=100.00  +MOVJ EC00088 VJ=100.00
'R-L Trip
MOVJ C00089 BC00089 VJ=100.00  +MOVJ EC00089 VJ=100.00
CALL JOB:CLEAN-R1_KM_NEW
'WireCut
MOVJ C00090 BC00090 VJ=100.00  +MOVJ EC00090 VJ=100.00
'Path S4234
SFTOF3D
MOVJ C00091 BC00091 VJ=100.00  +MOVJ EC00091 VJ=100.00
MOVL C00092 BC00092 V=800.0  +MOVJ EC00092 VJ=100.00
SMOVL C00093 BC00093 V=166.7  +MOVJ EC00093
SREFP 3 C00094 BC00094  +REFP EC00094
CALL JOB:SEARCH-R1-S13D
SET P034 P006
SFTON3D P034
SMOVL C00095 BC00095 V=166.7  +MOVJ EC00095
SMOVL C00096 BC00096 V=166.7  +MOVJ EC00096
SREFP 3 C00097 BC00097  +REFP EC00097
CALL JOB:SEARCH-R1-S13D
SET P034 P006
SFTON3D P034
SMOVL C00098 BC00098 V=166.7  +MOVJ EC00098
MOVL C00099 BC00099 V=800.0  +MOVJ EC00099 VJ=100.00
MOVL C00100 BC00100 V=1000.0  +MOVJ EC00100 VJ=100.00
'EndPath S4234
'Path S4235
SFTOF3D
MOVJ C00101 BC00101 VJ=100.00  +MOVJ EC00101 VJ=100.00
MOVL C00102 BC00102 V=800.0  +MOVJ EC00102 VJ=100.00
SMOVL C00103 BC00103 V=166.7  +MOVJ EC00103
SREFP 3 C00104 BC00104  +REFP EC00104
CALL JOB:SEARCH-R1-S13D
SET P033 P006
SFTON3D P033
SMOVL C00105 BC00105 V=166.7  +MOVJ EC00105
SMOVL C00106 BC00106 V=166.7  +MOVJ EC00106
SREFP 3 C00107 BC00107  +REFP EC00107
CALL JOB:SEARCH-R1-S13D
SET P033 P006
SFTON3D P033
SMOVL C00108 BC00108 V=166.7  +MOVJ EC00108
MOVL C00109 BC00109 V=800.0  +MOVJ EC00109 VJ=100.00
MOVL C00110 BC00110 V=1000.0  +MOVJ EC00110 VJ=100.00
'EndPath S4235
'Path S4236
SFTOF3D
MOVJ C00111 BC00111 VJ=100.00  +MOVJ EC00111 VJ=100.00
MOVL C00112 BC00112 V=800.0  +MOVJ EC00112 VJ=100.00
SMOVL C00113 BC00113 V=166.7  +MOVJ EC00113
SREFP 3 C00114 BC00114  +REFP EC00114
CALL JOB:SEARCH-R1-S13D
SET P024 P006
SFTON3D P024
SMOVL C00115 BC00115 V=166.7  +MOVJ EC00115
SMOVL C00116 BC00116 V=166.7  +MOVJ EC00116
SREFP 3 C00117 BC00117  +REFP EC00117
CALL JOB:SEARCH-R1-S13D
SET P024 P006
SFTON3D P024
SMOVL C00118 BC00118 V=166.7  +MOVJ EC00118
MOVL C00119 BC00119 V=800.0  +MOVJ EC00119 VJ=100.00
MOVL C00120 BC00120 V=1000.0  +MOVJ EC00120 VJ=100.00
'EndPath S4236
'Path S4237
SFTOF3D
MOVJ C00121 BC00121 VJ=100.00  +MOVJ EC00121 VJ=100.00
MOVL C00122 BC00122 V=800.0  +MOVJ EC00122 VJ=100.00
SMOVL C00123 BC00123 V=166.7  +MOVJ EC00123
SREFP 3 C00124 BC00124  +REFP EC00124
CALL JOB:SEARCH-R1-S13D
SET P023 P006
SFTON3D P023
SMOVL C00125 BC00125 V=166.7  +MOVJ EC00125
SMOVL C00126 BC00126 V=166.7  +MOVJ EC00126
SREFP 3 C00127 BC00127  +REFP EC00127
CALL JOB:SEARCH-R1-S13D
SET P023 P006
SFTON3D P023
SMOVL C00128 BC00128 V=166.7  +MOVJ EC00128
MOVL C00129 BC00129 V=800.0  +MOVJ EC00129 VJ=100.00
MOVL C00130 BC00130 V=1000.0  +MOVJ EC00130 VJ=100.00
'EndPath S4237
'nowe
'Path W4903
SFTOF3D
SFTON3D P024
MOVJ C00131 BC00131 VJ=100.00  +MOVJ EC00131 VJ=100.00
SMOVL C00132 BC00132 V=800.0  +MOVJ EC00132
SMOVL C00133 BC00133 V=150.0 PL=0  +MOVJ EC00133
MACRO1 MJ#(0) ARGF14
ARCON
SMOVL C00134 BC00134 V=9.2  +MOVJ EC00134
SFTON3D P023
SMOVL C00135 BC00135 V=9.2  +MOVJ EC00135
SMOVL C00136 BC00136 V=9.2  +MOVJ EC00136
ARCOF
SMOVL C00137 BC00137 V=800.0  +MOVJ EC00137
SMOVL C00138 BC00138 V=1000.0  +MOVJ EC00138
SFTOF3D
'EndPath W4903
'Path W4906
SFTOF3D
SFTON3D P033
MOVJ C00139 BC00139 VJ=100.00  +MOVJ EC00139 VJ=100.00
SMOVL C00140 BC00140 V=800.0  +MOVJ EC00140
SMOVL C00141 BC00141 V=150.0 PL=0  +MOVJ EC00141
ARCON
SFTON3D P034
SMOVL C00142 BC00142 V=10.7  +MOVJ EC00142
ARCOF
SMOVL C00143 BC00143 V=800.0  +MOVJ EC00143
SMOVL C00144 BC00144 V=1000.0  +MOVJ EC00144
SFTOF3D
'EndPath W4906
MOVJ C00145 BC00145 VJ=100.00  +MOVJ EC00145 VJ=100.00
'WireCut
MOVJ C00146 BC00146 VJ=100.00  +MOVJ EC00146 VJ=100.00
MOVJ C00147 BC00147 VJ=100.00  +MOVJ EC00147 VJ=100.00
MOVJ C00148 BC00148 VJ=100.00  +MOVJ EC00148 VJ=100.00
MOVJ C00149 BC00149 VJ=100.00  +MOVJ EC00149 VJ=100.00
CALL JOB:CLEAN-R1_KM_NEW
MOVJ C00150 BC00150 VJ=100.00  +MOVJ EC00150 VJ=100.00
MOVJ C00151 BC00151 VJ=100.00  +MOVJ EC00151 VJ=100.00
'L-R Trip
'Path S4249
SFTOF3D
MOVJ C00152 BC00152 VJ=100.00  +MOVJ EC00152 VJ=100.00
MOVL C00153 BC00153 V=800.0  +MOVJ EC00153 VJ=100.00
SMOVL C00154 BC00154 V=166.7  +MOVJ EC00154
SREFP 3 C00155 BC00155  +REFP EC00155
CALL JOB:SEARCH-R1-S13D
SET P036 P006
SFTON3D P036
SMOVL C00156 BC00156 V=166.7  +MOVJ EC00156
SMOVL C00157 BC00157 V=166.7  +MOVJ EC00157
SREFP 3 C00158 BC00158  +REFP EC00158
CALL JOB:SEARCH-R1-S13D
SET P036 P006
SFTON3D P036
SMOVL C00159 BC00159 V=166.7  +MOVJ EC00159
MOVL C00160 BC00160 V=800.0  +MOVJ EC00160 VJ=100.00
MOVL C00161 BC00161 V=1000.0  +MOVJ EC00161 VJ=100.00
'EndPath S4249
'Path S4250
SFTOF3D
MOVJ C00162 BC00162 VJ=100.00  +MOVJ EC00162 VJ=100.00
MOVL C00163 BC00163 V=800.0  +MOVJ EC00163 VJ=100.00
SMOVL C00164 BC00164 V=166.7  +MOVJ EC00164
SREFP 3 C00165 BC00165  +REFP EC00165
CALL JOB:SEARCH-R1-S13D
SET P035 P006
SFTON3D P035
SMOVL C00166 BC00166 V=166.7  +MOVJ EC00166
SMOVL C00167 BC00167 V=166.7  +MOVJ EC00167
SREFP 3 C00168 BC00168  +REFP EC00168
CALL JOB:SEARCH-R1-S13D
SET P035 P006
SFTON3D P035
SMOVL C00169 BC00169 V=166.7  +MOVJ EC00169
MOVL C00170 BC00170 V=800.0  +MOVJ EC00170 VJ=100.00
MOVL C00171 BC00171 V=1000.0  +MOVJ EC00171 VJ=100.00
'EndPath S4250
'Path S4251
SFTOF3D
MOVJ C00172 BC00172 VJ=100.00  +MOVJ EC00172 VJ=100.00
MOVL C00173 BC00173 V=800.0  +MOVJ EC00173 VJ=100.00
SMOVL C00174 BC00174 V=166.7  +MOVJ EC00174
SREFP 3 C00175 BC00175  +REFP EC00175
CALL JOB:SEARCH-R1-S13D
SET P026 P006
SFTON3D P026
SMOVL C00176 BC00176 V=166.7  +MOVJ EC00176
SMOVL C00177 BC00177 V=166.7  +MOVJ EC00177
SREFP 3 C00178 BC00178  +REFP EC00178
CALL JOB:SEARCH-R1-S13D
SET P026 P006
SFTON3D P026
SMOVL C00179 BC00179 V=166.7  +MOVJ EC00179
MOVL C00180 BC00180 V=800.0  +MOVJ EC00180 VJ=100.00
MOVL C00181 BC00181 V=1000.0  +MOVJ EC00181 VJ=100.00
'EndPath S4251
'Path S4252
SFTOF3D
MOVJ C00182 BC00182 VJ=100.00  +MOVJ EC00182 VJ=100.00
MOVL C00183 BC00183 V=800.0  +MOVJ EC00183 VJ=100.00
SMOVL C00184 BC00184 V=166.7  +MOVJ EC00184
SREFP 3 C00185 BC00185  +REFP EC00185
CALL JOB:SEARCH-R1-S13D
SET P025 P006
SFTON3D P025
SMOVL C00186 BC00186 V=166.7  +MOVJ EC00186
SMOVL C00187 BC00187 V=166.7  +MOVJ EC00187
SREFP 3 C00188 BC00188  +REFP EC00188
CALL JOB:SEARCH-R1-S13D
SET P025 P006
SFTON3D P025
SMOVL C00189 BC00189 V=166.7  +MOVJ EC00189
MOVL C00190 BC00190 V=800.0  +MOVJ EC00190 VJ=100.00
MOVL C00191 BC00191 V=1000.0  +MOVJ EC00191 VJ=100.00
'EndPath S4252
'Path W4907
SFTOF3D
SFTON3D P026
MOVJ C00192 BC00192 VJ=100.00  +MOVJ EC00192 VJ=100.00
SMOVL C00193 BC00193 V=800.0  +MOVJ EC00193
SMOVL C00194 BC00194 V=150.0 PL=0  +MOVJ EC00194
ARCON
SFTON3D P025
SMOVL C00195 BC00195 V=11.7  +MOVJ EC00195
ARCOF
SMOVL C00196 BC00196 V=800.0  +MOVJ EC00196
SMOVL C00197 BC00197 V=1000.0  +MOVJ EC00197
SFTOF3D
'EndPath W4907
'Path W4908
SFTOF3D
SFTON3D P035
MOVJ C00198 BC00198 VJ=100.00  +MOVJ EC00198 VJ=100.00
SMOVL C00199 BC00199 V=800.0  +MOVJ EC00199
SMOVL C00200 BC00200 V=150.0 PL=0  +MOVJ EC00200
ARCON
SFTON3D P036
SMOVL C00201 BC00201 V=11.7  +MOVJ EC00201
ARCOF
SMOVL C00202 BC00202 V=800.0  +MOVJ EC00202
SMOVL C00203 BC00203 V=1000.0  +MOVJ EC00203
SFTOF3D
'EndPath W4908
MOVJ C00204 BC00204 VJ=100.00  +MOVJ EC00204 VJ=100.00
MOVJ C00205 BC00205 VJ=100.00  +MOVJ EC00205 VJ=100.00
CALL JOB:CLEAN-R1_KM_NEW
MOVJ C00206 BC00206 VJ=100.00  +MOVJ EC00206 VJ=100.00
MOVJ C00207 BC00207 VJ=100.00  +MOVJ EC00207 VJ=100.00
MOVJ C00208 BC00208 VJ=100.00  +MOVJ EC00208 VJ=100.00
'Path S4888
SFTOF3D
MOVJ C00209 BC00209 VJ=100.00  +MOVJ EC00209 VJ=100.00
MOVL C00210 BC00210 V=800.0  +MOVJ EC00210 VJ=100.00
SMOVL C00211 BC00211 V=166.7  +MOVJ EC00211
SREFP 3 C00212 BC00212  +REFP EC00212
CALL JOB:SEARCH-R1-S13D
SET P044 P006
SFTON3D P044
SMOVL C00213 BC00213 V=166.7  +MOVJ EC00213
SMOVL C00214 BC00214 V=166.7  +MOVJ EC00214
SREFP 3 C00215 BC00215  +REFP EC00215
CALL JOB:SEARCH-R1-S13D
SET P044 P006
SFTON3D P044
SMOVL C00216 BC00216 V=166.7  +MOVJ EC00216
MOVL C00217 BC00217 V=800.0  +MOVJ EC00217 VJ=100.00
MOVL C00218 BC00218 V=1000.0  +MOVJ EC00218 VJ=100.00
'EndPath S4888
'Path S4889
SFTOF3D
MOVJ C00219 BC00219 VJ=100.00  +MOVJ EC00219 VJ=100.00
MOVL C00220 BC00220 V=800.0  +MOVJ EC00220 VJ=100.00
SMOVL C00221 BC00221 V=166.7  +MOVJ EC00221
SREFP 3 C00222 BC00222  +REFP EC00222
CALL JOB:SEARCH-R1-S13D
SET P043 P006
SFTON3D P043
SMOVL C00223 BC00223 V=166.7  +MOVJ EC00223
SMOVL C00224 BC00224 V=166.7  +MOVJ EC00224
SREFP 3 C00225 BC00225  +REFP EC00225
CALL JOB:SEARCH-R1-S13D
SET P043 P006
SFTON3D P043
SMOVL C00226 BC00226 V=166.7  +MOVJ EC00226
MOVL C00227 BC00227 V=800.0  +MOVJ EC00227 VJ=100.00
MOVL C00228 BC00228 V=1000.0  +MOVJ EC00228 VJ=100.00
'EndPath S4889
MOVJ C00229 BC00229 VJ=100.00  +MOVJ EC00229 VJ=100.00
MOVJ C00230 BC00230 VJ=100.00  +MOVJ EC00230 VJ=100.00
MOVJ C00231 BC00231 VJ=100.00  +MOVJ EC00231 VJ=100.00
MOVJ C00232 BC00232 VJ=100.00  +MOVJ EC00232 VJ=100.00
'Path S4899
SFTOF3D
MOVJ C00233 BC00233 VJ=100.00  +MOVJ EC00233 VJ=100.00
MOVL C00234 BC00234 V=800.0  +MOVJ EC00234 VJ=100.00
SMOVL C00235 BC00235 V=166.7  +MOVJ EC00235
SREFP 3 C00236 BC00236  +REFP EC00236
CALL JOB:SEARCH-R1-S13D
SET P046 P006
SFTON3D P046
SMOVL C00237 BC00237 V=166.7  +MOVJ EC00237
SMOVL C00238 BC00238 V=166.7  +MOVJ EC00238
SREFP 3 C00239 BC00239  +REFP EC00239
CALL JOB:SEARCH-R1-S13D
SET P046 P006
SFTON3D P046
SMOVL C00240 BC00240 V=166.7  +MOVJ EC00240
MOVL C00241 BC00241 V=800.0  +MOVJ EC00241 VJ=100.00
MOVL C00242 BC00242 V=1000.0  +MOVJ EC00242 VJ=100.00
'EndPath S4899
MOVJ C00243 BC00243 VJ=100.00  +MOVJ EC00243 VJ=100.00
'Path S4888
SFTOF3D
MOVJ C00244 BC00244 VJ=100.00  +MOVJ EC00244 VJ=100.00
MOVL C00245 BC00245 V=800.0  +MOVJ EC00245 VJ=100.00
SMOVL C00246 BC00246 V=166.7  +MOVJ EC00246
SREFP 3 C00247 BC00247  +REFP EC00247
CALL JOB:SEARCH-R1-S13D
SET P028 P006
SFTON3D P028
SMOVL C00248 BC00248 V=166.7  +MOVJ EC00248
SMOVL C00249 BC00249 V=166.7  +MOVJ EC00249
SREFP 3 C00250 BC00250  +REFP EC00250
CALL JOB:SEARCH-R1-S13D
SET P028 P006
SFTON3D P028
SMOVL C00251 BC00251 V=166.7  +MOVJ EC00251
MOVL C00252 BC00252 V=800.0  +MOVJ EC00252 VJ=100.00
MOVL C00253 BC00253 V=1000.0  +MOVJ EC00253 VJ=100.00
'EndPath S4888
'Path S4889
SFTOF3D
MOVJ C00254 BC00254 VJ=100.00  +MOVJ EC00254 VJ=100.00
MOVL C00255 BC00255 V=800.0  +MOVJ EC00255 VJ=100.00
SMOVL C00256 BC00256 V=166.7  +MOVJ EC00256
SREFP 3 C00257 BC00257  +REFP EC00257
CALL JOB:SEARCH-R1-S13D
SET P027 P006
SFTON3D P027
SMOVL C00258 BC00258 V=166.7  +MOVJ EC00258
SMOVL C00259 BC00259 V=166.7  +MOVJ EC00259
SREFP 3 C00260 BC00260  +REFP EC00260
CALL JOB:SEARCH-R1-S13D
SET P027 P006
SFTON3D P027
SMOVL C00261 BC00261 V=166.7  +MOVJ EC00261
MOVL C00262 BC00262 V=800.0  +MOVJ EC00262 VJ=100.00
MOVL C00263 BC00263 V=1000.0  +MOVJ EC00263 VJ=100.00
'EndPath S4889
'Path W4890
SFTOF3D
SFTON3D P027
MOVJ C00264 BC00264 VJ=100.00  +MOVJ EC00264 VJ=100.00
SMOVL C00265 BC00265 V=800.0  +MOVJ EC00265
SMOVL C00266 BC00266 V=150.0 PL=0  +MOVJ EC00266
MACRO1 MJ#(0) ARGF6
ARCON
SMOVL C00267 BC00267 V=6.7  +MOVJ EC00267
SFTON3D P028
SMOVL C00268 BC00268 V=10.0  +MOVJ EC00268
ARCOF
SMOVL C00269 BC00269 V=800.0  +MOVJ EC00269
SMOVL C00270 BC00270 V=1000.0  +MOVJ EC00270
SFTOF3D
'EndPath W4890
MOVJ C00271 BC00271 VJ=100.00  +MOVJ EC00271 VJ=100.00
MOVJ C00272 BC00272 VJ=100.00  +MOVJ EC00272 VJ=100.00
MOVJ C00273 BC00273 VJ=100.00  +MOVJ EC00273 VJ=100.00
MOVJ C00274 BC00274 VJ=100.00  +MOVJ EC00274 VJ=100.00
MOVJ C00275 BC00275 VJ=100.00  +MOVJ EC00275 VJ=100.00
'Path W4900
SFTOF3D
SFTON3D P043
MOVJ C00276 BC00276 VJ=100.00  +MOVJ EC00276 VJ=100.00
SMOVL C00277 BC00277 V=800.0  +MOVJ EC00277
SMOVL C00278 BC00278 V=150.0 PL=0  +MOVJ EC00278
MACRO1 MJ#(0) ARGF14
ARCON
SFTON3D P044
SMOVL C00279 BC00279 V=10.0  +MOVJ EC00279
SMOVL C00280 BC00280 V=10.0  +MOVJ EC00280
ARCOF
SMOVL C00281 BC00281 V=800.0  +MOVJ EC00281
SMOVL C00282 BC00282 V=1000.0  +MOVJ EC00282
SFTOF3D
'EndPath W4900
MOVJ C00283 BC00283 VJ=100.00  +MOVJ EC00283 VJ=100.00
MOVJ C00284 BC00284 VJ=100.00  +MOVJ EC00284 VJ=100.00
MOVJ C00285 BC00285 VJ=100.00  +MOVJ EC00285 VJ=100.00
MOVJ C00286 BC00286 VJ=100.00  +MOVJ EC00286 VJ=100.00
MOVJ C00287 BC00287 VJ=100.00  +MOVJ EC00287 VJ=100.00
'Path W4898
SFTOF3D
SFTON3D P046
MOVJ C00288 BC00288 VJ=100.00  +MOVJ EC00288 VJ=100.00
SMOVL C00289 BC00289 V=800.0  +MOVJ EC00289
SMOVL C00290 BC00290 V=150.0 PL=0  +MOVJ EC00290
ARCON
SMOVL C00291 BC00291 V=10.0  +MOVJ EC00291
SMOVL C00292 BC00292 V=10.0  +MOVJ EC00292
ARCOF
SMOVL C00293 BC00293 V=800.0  +MOVJ EC00293
SMOVL C00294 BC00294 V=1000.0  +MOVJ EC00294
SFTOF3D
'EndPath W4898
MOVJ C00295 BC00295 VJ=100.00  +MOVJ EC00295 VJ=100.00
MOVJ C00296 BC00296 VJ=100.00  +MOVJ EC00296 VJ=100.00
MOVJ C00297 BC00297 VJ=100.00  +MOVJ EC00297 VJ=100.00
MOVJ C00298 BC00298 VJ=100.00  +MOVJ EC00298 VJ=100.00
MOVJ C00299 BC00299 VJ=100.00  +MOVJ EC00299 VJ=100.00
END
